ABB RobotStudio station: Welding Routine.rspag

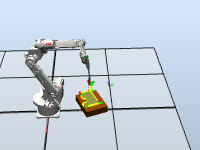
--- station ---
Station Welding (saved by RobotStudio 6.6.7688.1025)
Controller System3
  mechanical unit ROB_1: IRB1520ID_4_150__02, 6 joints, base frame (0, 0, 0) mm
Layout (positions relative to the parent item):
  - IRB1520ID_4_150__02 [mechanism, from Robots\IRB1520ID_4_150_G_02.rslib] at (0, 0, 0) mm; joint values [1.3508, -0.5618, 0.4308, -0.5213, 1.3433, 1.0164] (rad or m)
  - Curve_thing [part, from Training Objects\Curve_Thing.rslib] at (491.71, 446.12, 553.55) mm, rotated rx 0.75 ry 0.87 rz 20.92 deg
  - RA_MTG4000_22 [mechanism, from Tools\Fronius_Robacta_MTG4000_22deg.rslib] at (226.3, 567.45, 1083.41) mm, rotated rx 179.07 ry 36.08 rz -159.64 deg
Attachment: RA_MTG4000_22 is attached to IRB1520ID_4_150__02 / Link6

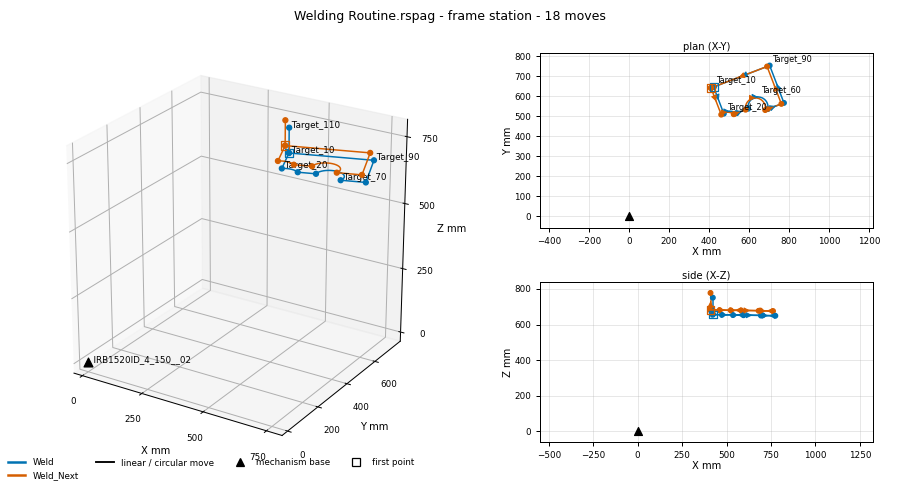
[picture p0: tool path of Welding Routine.rspag in frame station, 18 of 18 moves have a stored position in this frame; points joined in program order, loops and branches not executed]
--- Backups/System3/RAPID/TASK1/PROGMOD/CalibData.mod ---
MODULE CalibData
	PERS tooldata Weldgun:=[TRUE,[[20.31,0,363.689],[0.948464781,0,0.316882565,0]],[1,[0,0,1],[1,0,0,0],0,0,0]];
	TASK PERS wobjdata Wobj_CurveThing:=[FALSE,TRUE,"",[[-864.223701906,1007.902511198,-127.503563299],[0.967349797,0.10345319,-0.213524278,-0.089102138]],[[0,0,0],[1,0,0,0]]];
ENDMODULE

--- Backups/System3/RAPID/TASK1/PROGMOD/Module1.mod ---
MODULE Module1
	CONST robtarget Target_10:=[[1536.576556246,3.869682319,198.770937231],[0.237551598,0.2611991,-0.93374636,0.058838794],[0,0,0,0],[9E+09,9E+09,9E+09,9E+09,9E+09,9E+09]];
	CONST robtarget Target_20:=[[1610.262431772,-118.519517981,196.739917302],[0.237551598,0.2611991,-0.93374636,0.058838794],[0,0,0,0],[9E+09,9E+09,9E+09,9E+09,9E+09,9E+09]];
	CONST robtarget Target_30:=[[1635.06425627,-103.151208524,181.020759767],[0.237551598,0.2611991,-0.93374636,0.058838794],[0,0,0,0],[9E+09,9E+09,9E+09,9E+09,9E+09,9E+09]];
	CONST robtarget Target_40:=[[1665.177493119,-108.87059946,168.415646466],[0.237551598,0.2611991,-0.93374636,0.058838794],[0,0,0,0],[9E+09,9E+09,9E+09,9E+09,9E+09,9E+09]];
	CONST robtarget Target_50:=[[1712.786308837,-79.707904703,138.33144096],[0.237551598,0.2611991,-0.93374636,0.058838794],[0,0,0,0],[9E+09,9E+09,9E+09,9E+09,9E+09,9E+09]];
	CONST robtarget Target_60:=[[1744.603044356,-16.849387742,106.697958569],[0.237551598,0.2611991,-0.93374636,0.058838794],[0,0,0,0],[9E+09,9E+09,9E+09,9E+09,9E+09,9E+09]];
	CONST robtarget Target_70:=[[1800.020788346,-69.266593363,94.636232832],[0.237551598,0.2611991,-0.93374636,0.058838794],[0,0,0,0],[9E+09,9E+09,9E+09,9E+09,9E+09,9E+09]];
	CONST robtarget Target_80:=[[1864.931500786,-29.505652771,53.618887974],[0.237551598,0.2611991,-0.93374636,0.058838794],[0,0,0,0],[9E+09,9E+09,9E+09,9E+09,9E+09,9E+09]];
	CONST robtarget Target_90:=[[1761.783117483,141.819557854,56.46198946],[0.237551598,0.2611991,-0.93374636,0.058838794],[0,0,0,0],[9E+09,9E+09,9E+09,9E+09,9E+09,9E+09]];
	CONST robtarget Target_100:=[[1536.576556246,3.869682319,198.770937231],[0.237551598,0.2611991,-0.93374636,0.058838794],[0,0,0,0],[9E+09,9E+09,9E+09,9E+09,9E+09,9E+09]];
    CONST robtarget Target_110:=[[1573.94382832,26.42268631,282.790606684],[0.237551462,0.261199153,-0.933746385,0.058838711],[0,-1,0,0],[9E+09,9E+09,9E+09,9E+09,9E+09,9E+09]];

	! This function starts welding the work object
    PROC Weld()
	    MoveL Target_10,v80,z0,Weldgun\WObj:=Wobj_CurveThing;
	    MoveL Target_20,v80,z0,Weldgun\WObj:=Wobj_CurveThing;
	    MoveC Target_30,Target_40,v80,z0,Weldgun\WObj:=Wobj_CurveThing;
	    MoveL Target_50,v80,z0,Weldgun\WObj:=Wobj_CurveThing;
	    MoveC Target_60,Target_70,v80,z0,Weldgun\WObj:=Wobj_CurveThing;
	    MoveL Target_80,v80,z0,Weldgun\WObj:=Wobj_CurveThing;
	    MoveL Target_90,v80,z0,Weldgun\WObj:=Wobj_CurveThing;
	    MoveL Target_100,v80,z0,Weldgun\WObj:=Wobj_CurveThing;
        MoveL Target_110,v80,z0,Weldgun\WObj:=Wobj_CurveThing;
        WaitTime 3; ! Waits 3 second to place another work object
        Weld_Next; ! Calls the function to weld the next workobject
	ENDPROC

    ! This function starts welding the next work object
    PROC Weld_Next()
        MoveL offs(Target_10,0,0,30),v80,z0,Weldgun\WObj:=Wobj_CurveThing;
	    MoveL offs(Target_20,0,0,30),v80,z0,Weldgun\WObj:=Wobj_CurveThing;
	    MoveC offs(Target_30,0,0,30), offs(Target_40,0,0,30),v80,z0,Weldgun\WObj:=Wobj_CurveThing;
	    MoveL offs(Target_50,0,0,30),v80,z0,Weldgun\WObj:=Wobj_CurveThing;
	    MoveC offs(Target_60,0,0,30), offs(Target_70,0,0,30),v80,z0,Weldgun\WObj:=Wobj_CurveThing;
	    MoveL offs(Target_80,0,0,30),v80,z0,Weldgun\WObj:=Wobj_CurveThing;
	    MoveL offs(Target_90,0,0,30),v80,z0,Weldgun\WObj:=Wobj_CurveThing;
	    MoveL offs(Target_100,0,0,30),v80,z0,Weldgun\WObj:=Wobj_CurveThing;
        MoveL offs(Target_110,0,0,30),v80,z0,Weldgun\WObj:=Wobj_CurveThing;
    ENDPROC

ENDMODULE

--- Backups/System3/RAPID/TASK1/SYSMOD/LINKEDM.sys ---
%%%
  VERSION:1
  LANGUAGE:ENGLISH
%%%

MODULE LINKEDM (SYSMODULE)

! FOLLOWER
!     Name of electronically linked follower axis used by operator at teach pendent.
      PERS string l_f_axis_name{5}       :=  ["",  "", "", "", ""];

!     Name of the mechanical unit for follower axis.
      PERS string l_f_mecunt_n{5}  :=  ["", "", "", "", ""];

!     Linked follower axis number in the mechanical unit (first axis in mech. unit is number 1).
      PERS num l_f_axis_no{5}      :=  [0,          0,   0,  0,  0];

! MASTER
!     Name of the mechanical unit for linked master axis.
      PERS string l_m_mecunt_n{5} :=  ["", "", "", "", ""];

!     Linked master axis number in the mechanical unit (first axis in mech. unit is number 1).
!     See axis number table in documentation for different master mechanical units.
      PERS num l_m_axis_no{5}     :=  [0,  0,  0,  0,  0];

! POSITION OFFSET
!     The increase of the allowed offset position between the master and follower
!     positions, used when starting AUTO mode. As soon as the offset is decreased
!     the old configurated parameter is used.
!     Example: 3 => the configurated value of allowed offset is increased 3 times.
      PERS num offset_ratio{5}       :=  [10,  10,   10,  10,  10];

! SPEED RATIO
!     Speed_ratio used in AUTO and JOG modes [ very_slow   slow    normal    fast]
!     Value 1 = max allowed manual speed.
      CONST num speed_ratio {20}      := [0.01, 0.01, 0.01, 0.01, 0.01,
                                          0.05, 0.05, 0.05, 0.05, 0.05,
                                          0.20, 0.20, 0.20, 0.20, 0.20,
                                          1.00, 1.00, 1.00, 1.00, 1.00];

! STEP SIZE
!     Displacement position used in JOG mode for each activation of positive or
!     negative movement.                  [very_short    short   normal   long]
!     Unit degees or meter.
      CONST num displacement {20}     := [0.001, 0.001, 0.001, 0.001, 0.001,
                                          0.005, 0.005, 0.005, 0.005, 0.005,
                                          0.020, 0.020, 0.020, 0.020, 0.020,
                                          0.100, 0.100, 0.100, 0.100, 0.100];


!-------------------------------------------------------------
 PROC Linked_m ()
      Linked_m_exe ;
 ENDPROC
ENDMODULE
